// TIA Portal V15.1 export
// export: Created 2024-06-21T08:40:51.1181016Z, ExportSetting WithDefaults, DisplayName Totally Integrated Automation Portal, DisplayVersion V15.1 Update 5, DisplayName TIA Portal Openness, DisplayVersion V15.1 Update 5, DisplayName SINAMICS Startdrive Advanced, DisplayVersion V15.1, DisplayName G130, G150, S120, S150, SINAMICS MV, S210, DisplayVersion V15.1, DisplayName G110M, G120, G120C, G120D, G120P, DisplayVersion V15.1, DisplayName STEP 7 Professional, DisplayVersion V15.1 Update 5, DisplayName STEP 7 Safety, DisplayVersion V15.1, DisplayName WinCC Professional, DisplayVersion V15.1 Update 5, DisplayName SIMATIC Visualization Architect, DisplayVersion V15.1
DATA_BLOCK "_209230ZM01Config"   // DB402
{ S7_Optimized_Access := 'FALSE' }
AUTHOR : VCC
VERSION : 0.1
// stored: AutoNumber false, DBAccessibleFromOPCUA true, IsOnlyStoredInLoadMemory false, IsWriteProtectedInAS false
   VAR
      Andon { ExternalAccessible := 'False'; ExternalVisible := 'False'; ExternalWritable := 'False'} : "AndonConfigVCG";   // Config
      "230CHB21" { ExternalAccessible := 'False'; ExternalVisible := 'False'; ExternalWritable := 'False'} : "MovUnit2Pos2S-MoviFitFCPNConfig";   // Config
      "230CHB22" { ExternalAccessible := 'False'; ExternalVisible := 'False'; ExternalWritable := 'False'} : "MovUnit2Pos2S-MoviFitFCPNConfig";   // Config
      "230CA21" { ExternalAccessible := 'False'; ExternalVisible := 'False'; ExternalWritable := 'False'} : "RollerConvMoviFitFCPNConfig";   // Config
      "230CR22" { ExternalAccessible := 'False'; ExternalVisible := 'False'; ExternalWritable := 'False'} : "RollerConvMoviFitFCPNConfig";   // Config
      "230ASH01" { ExternalAccessible := 'False'; ExternalVisible := 'False'; ExternalWritable := 'False'} : "HandHeldHBA-Config";   // Config
   END_VAR
BEGIN
END_DATA_BLOCK
